{attribute 'linkalways'} 
{attribute 'no_explicit_call' := 'This FB is a CLASS and must be accessed using methods or properties'}
{attribute 'enable_dynamic_creation'}
FUNCTION_BLOCK _Array0to10OfBool EXTENDS ArrayDatatypeBase
VAR CONSTANT
	lBound : DINT := 0;
	uBound : DINT := 10;
END_VAR
VAR
	localData : ARRAY [lBound..uBound] OF BOOL;
	activeData : REFERENCE TO ARRAY [lBound..uBound] OF BOOL REF= localData;
	elements : ARRAY [lBound..uBound] OF _BOOL(FALSE);
	baseType : _BOOL(FALSE);
END_VAR

PROPERTY PUBLIC Address : PVOID
GET
Address := ADR(activeData);
END_GET
END_PROPERTY

PROPERTY PUBLIC BaseDatatype : I_Datatype
GET
BaseDatatype := baseType;
END_GET
END_PROPERTY

METHOD PUBLIC ClearReference
VAR_INPUT
END_VAR
activeData REF= localData;
SetElementReference();
END_METHOD

METHOD PUBLIC Clone : I_Datatype
VAR
    pClone : POINTER TO _Array0to10OfBool;
END_VAR
pClone := __NEW(_Array0to10OfBool());
pClone^.Value := Value;
Clone := pClone^;
END_METHOD

METHOD FB_init : BOOL
VAR_INPUT
	bInitRetains : BOOL; // if TRUE, the retain variables are initialized (warm start / cold start)
	bInCopyCode : BOOL;  // if TRUE, the instance afterwards gets moved into the copy code (online change)
END_VAR
SetElementReference();
END_METHOD

METHOD PUBLIC GetElementAsDatatypeByIndex : I_Datatype
VAR_INPUT
	Index : DINT;
END_VAR
GetElementAsDatatypeByIndex := elements[Index];
END_METHOD

METHOD PUBLIC GetElementByIndex : REFERENCE TO _BOOL;
VAR_INPUT
	Index : DINT;
END_VAR
GetElementByIndex REF= elements[Index];
END_METHOD

PROPERTY PUBLIC LowerBound : DINT
GET
LowerBound := lBound;
END_GET
END_PROPERTY

METHOD PUBLIC MakeReferenceTo
VAR_INPUT
	ReferenceTarget : REFERENCE TO ARRAY [lBound..uBound] OF BOOL;
END_VAR
activeData REF= ReferenceTarget;
SetElementReference();
END_METHOD

METHOD PROTECTED OnSerializeArrayValues
VAR_INPUT
	Serializer : I_Serializer;
END_VAR
VAR
	i : DINT;
END_VAR
FOR i := lBound TO uBound DO
	elements[i].SerializeWith(Serializer);
END_FOR
END_METHOD

METHOD PROTECTED SetElementReference
VAR_INPUT
END_VAR
VAR
	i : DINT;
END_VAR
FOR i := lBound TO uBound DO
	elements[i].MakeReferenceTo(activeData[i]);
END_FOR
END_METHOD

PROPERTY PUBLIC Size : UDINT
GET
Size := SIZEOF(activeData);
END_GET
END_PROPERTY

METHOD PROTECTED TryDeserializeArrayValues : BOOL
VAR_INPUT
	Deserializer : I_Deserializer;
	Feedback : I_DeserializerFeedback;
END_VAR
VAR
	enumerator : I_DeserializerArrayForwardEnumerator;
	i : DINT;
END_VAR
enumerator := Deserializer.GetArrayEnumerator();
i := lBound;

WHILE enumerator.MoveNext() AND i <= uBound DO
	
	IF NOT elements[i].TryDeserializeFrom(enumerator.Current, Feedback) THEN
		EXIT;
	END_IF
	i := i + 1;

END_WHILE
enumerator.Dispose();
END_METHOD

METHOD TryMakeReferenceTo : BOOL
VAR_INPUT
	Target : I_Datatype;
END_VAR
VAR
	targetAsArray : I_ArrayDatatype;
	pTargetData : POINTER TO ARRAY [lBound..uBound] OF BOOL;
END_VAR
IF NOT Target.TryResolveAsArrayDatatype(targetAsArray) THEN
	RETURN;
END_IF

IF NOT (targetAsArray.Identifier = Identifier) THEN
	RETURN;
END_IF

pTargetData := Target.Address;
activeData REF= pTargetData^;
SetElementReference();
TryMakeReferenceTo := TRUE;
END_METHOD

PROPERTY PUBLIC UpperBound : DINT
GET
UpperBound := ubound;
END_GET
END_PROPERTY

PROPERTY PUBLIC Value : REFERENCE TO ARRAY [lBound..uBound] OF BOOL;
GET
Value ref= activeData;
END_GET
END_PROPERTY

END_FUNCTION_BLOCK

(* stored: Version 1.1.0.1, ProductVersion 3.1.4024.13
   POU _Array0to10OfBool: Id {4a9127d4-c160-08fd-0a37-72eed4d23ca2}, SpecialFunc None
   Folder Core: Id {9afbe3cc-1cc2-00a5-2da8-3e4bdffc8a57}
   Folder Constructor: Id {3a909e8b-446b-09af-12d8-17f0fec007ed}
   Folder Protected: Id {e6ce3210-7a14-0881-3983-4f79802ddd29}
   Folder Customize: Id {49b53497-65a8-0c29-1132-fb291828720e}
   Property Address: Id {70c960a5-aee0-09f4-05a9-8fb1350cf0ff}
   Get Get: Id {a40d98c1-4de4-02ce-0a96-a0be533abcf4}
   Property BaseDatatype: Id {e91c9b1f-0537-00c7-0845-64ac2d8bf358}
   Get Get: Id {4c6c4db1-d42c-02eb-3836-95a1f0bbc8b9}
   Method ClearReference: Id {d0595f49-17cf-0658-1d03-9817d0a92100}
   Method Clone: Id {e812f2ea-f547-0db0-05e5-9ad0ac9704dd}
   Method FB_init: Id {07aedd3a-6fb9-0f63-00af-ad2d481eed30}
   Method GetElementAsDatatypeByIndex: Id {0e15c8a3-ac86-0453-1aa9-31ad52185d0a}
   Method GetElementByIndex: Id {1db27bc8-4e7c-0628-0a26-3e61e166422e}
   Property LowerBound: Id {7880edb5-fa2d-0dac-0553-1fefd03d44b2}
   Get Get: Id {9fe561bb-b566-0924-262b-578d820a79c5}
   Method MakeReferenceTo: Id {d0a78fa8-7fe0-0693-27ec-da41958b77f5}
   Method OnSerializeArrayValues: Id {d3628e80-f909-0ba2-0d40-87567140c849}
   Method SetElementReference: Id {7bb7ade1-2f74-40d1-b6a8-94a495ce14c0}
   Property Size: Id {737987eb-8bbe-085c-1f73-fe25659fb1bd}
   Get Get: Id {714e6fe1-92a9-0213-3996-5615d074d98f}
   Method TryDeserializeArrayValues: Id {c3771a74-23bd-0e09-2997-a1f8bc83c542}
   Method TryMakeReferenceTo: Id {676573ad-8190-0c1c-0994-1de5ee38038f}
   Property UpperBound: Id {8476f69f-54ec-044d-047e-159700f17da9}
   Get Get: Id {7a4d714b-75a5-0c31-2bae-933caa3b9300}
   Property Value: Id {62685bbd-adad-0b40-3f91-5aaf07a0015c}
   Get Get: Id {389f4ae4-1592-0854-2c8b-4d3d3ce64b60} *)
